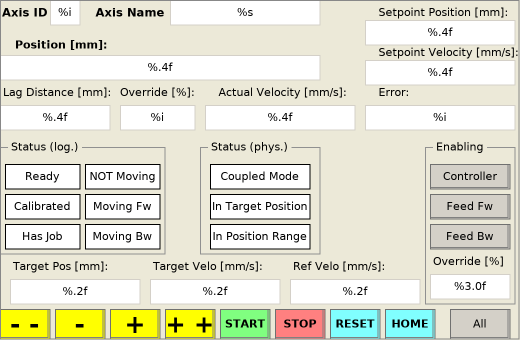
VISUALIZATION PH_NcAxis  // 520x340
VAR_IN_OUT
	stMcAxisOnline			: ST_McAxisOnline;	
END_VAR
    Group (0,0 320x25)
        Label (0,0 50x25), "Axis ID"
        Textfield (50,0 30x25), "%i", text variable: stMcAxisOnline.stStatus.dwAxisId
        Label (90,0 80x25), "Axis Name"
        Textfield (170,0 150x25), "%s", text variable: stMcAxisOnline.stStatus.sAxisName
    GroupBox (425,139 90x165), "Enabling"
        Button (5,25 80x25), "Controller", pressed state: stMcAxisOnline.mcPower.bEnable
            toggle stMcAxisOnline.mcPower.bEnable
        Button (5,85 80x25), "Feed Bw", pressed state: stMcAxisOnline.mcPower.bEnable_Negative
            toggle stMcAxisOnline.mcPower.bEnable_Negative
        Button (5,55 80x25), "Feed Fw", pressed state: stMcAxisOnline.mcPower.bEnable_Positive
            toggle stMcAxisOnline.mcPower.bEnable_Positive
        Textfield (5,135 80x25), "%3.0f", text variable: stMcAxisOnline.mcPower.lrOverride
            OnMouseClick: write the text variable via InputWithLimits, min 0, max 100
        Label (5,110 80x25), "Override [%]"
    Group (0,30 320x50)
        Textfield (0,25 320x25), "%.4f", text variable: stMcAxisOnline.stStatus.lrActPos
        Label (0,0 139x30), "Position [mm]:"
    GroupBox (200,139 120x115), "Status (phys.)"
        Rectangle (10,25 100x25), "Coupled Mode", colour toggle: stMcAxisOnline.stStatus.stAxisStatus.ProtectedMode
        Rectangle (10,55 100x25), "In Target Position", colour toggle: stMcAxisOnline.stStatus.stAxisStatus.InTargetPosition
        Rectangle (10,85 100x25), "In Position Range", colour toggle: stMcAxisOnline.stStatus.stAxisStatus.InPositionArea
    GroupBox (0,139 165x115), "Status (log.)"
        Rectangle (5,55 75x25), "Calibrated", colour toggle: stMcAxisOnline.stStatus.stAxisStatus.Homed
        Rectangle (5,85 75x25), "Has Job", colour toggle: stMcAxisOnline.stStatus.stAxisStatus.HasJob
        Rectangle (85,25 75x25), "NOT Moving", colour toggle: stMcAxisOnline.stStatus.stAxisStatus.NotMoving
        Rectangle (85,55 75x25), "Moving Fw", colour toggle: stMcAxisOnline.stStatus.stAxisStatus.PositiveDirection
        Rectangle (85,85 75x25), "Moving Bw", colour toggle: stMcAxisOnline.stStatus.stAxisStatus.NegativeDirection
        Rectangle (5,25 75x25), "Ready", colour toggle: stMcAxisOnline.stStatus.stAxisStatus.Operational
    Group (365,0 150x130)
        Label (0,0 150x25), "Setpoint Position [mm]:"
        Textfield (0,20 150x25), "%.4f", text variable: stMcAxisOnline.stStatus.lrSetPos
        Label (0,40 150x25), "Setpoint Velocity [mm/s]:"
        Textfield (0,60 150x25), "%.4f", text variable: stMcAxisOnline.stStatus.lrSetVelo
        Label (0,80 150x25), "Error:"
        Textfield (0,105 150x25), "%i", text variable: stMcAxisOnline.stStatus.udiNcErrorCode, colour toggle: stMcAxisOnline.stStatus.udiNcErrorCode>0
    Group (205,80 150x50)
        Label (0,0 150x25), "Actual Velocity [mm/s]:"
        Textfield (0,25 150x25), "%.4f", text variable: stMcAxisOnline.stStatus.lrActVelo
    Group (0,80 110x50)
        Label (0,0 110x25), "Lag Distance [mm]:"
        Textfield (0,25 110x25), "%.4f", text variable: stMcAxisOnline.stStatus.lrPosDiff
    Group (120,80 75x50)
        Label (0,0 75x25), "Override [%]:"
        Textfield (0,25 75x25), "%i", text variable: stMcAxisOnline.mcPower.lrOverride
    Group (10,254 410x50)
        Label (280,0 130x25), "Ref Velo [mm/s]:"
        Textfield (280,25 130x25), "%.2f", text variable: stMcAxisOnline.stAxisParameter.fDriveVeloReferenz
            OnMouseClick: write the text variable via Edit
        Label (0,0 130x25), "Target Pos [mm]:"
        Textfield (0,25 130x25), "%.2f", text variable: stMcAxisOnline.mcMoveAbsolute.lrPosition
            OnMouseClick: write the text variable via Edit
        Label (140,0 130x25), "Target Velo [mm/s]:"
        Textfield (140,25 130x25), "%.2f", text variable: stMcAxisOnline.mcMoveAbsolute.lrVelocity
            OnMouseClick: write the text variable via Edit
    Button (450,309 60x30), "All"
        OnMouseClick: execute {
            stMcAxisOnline.mcPower.bEnable				:= TRUE;
            stMcAxisOnline.mcPower.bEnable_Positive		:= TRUE;
            stMcAxisOnline.mcPower.bEnable_Negative		:= TRUE;
            stMcAxisOnline.mcPower.lrOverride			:= 100.0;
        }
    Group (0,309 435x30)
        Button (220,0 50x30), "START"
            tap stMcAxisOnline.mcMoveAbsolute.bExecute
        Button (275,0 50x30), "STOP"
            tap stMcAxisOnline.mcStop.bExecute
        Button (385,0 50x30), "HOME"
            tap stMcAxisOnline.mcHome.bExecute
        Button (330,0 50x30), "RESET"
            tap stMcAxisOnline.mcReset.bExecute
        Button (110,0 50x30), "+"
            tap stMcAxisOnline.mcJog.bSlowForward
        Button (165,0 50x30), "+ +"
            tap stMcAxisOnline.mcJog.bFastForward
        Button (55,0 50x30), "-"
            tap stMcAxisOnline.mcJog.bSlowBackward
        Button (0,0 50x30), "- -"
            tap stMcAxisOnline.mcJog.bFastBackward
END_VISUALIZATION

(* stored: Version 1.1.0.1, ProductVersion 3.1.4024.4
   Visu PH_NcAxis: Id {ef639a20-509b-44a6-b92e-e05f5e2f4660} *)
